{attribute 'OPC.UA.DA.StructuredType' := '1'}
{attribute 'OPC.UA.DA' := '1'}
TYPE stCombineAxisStatus :
STRUCT
    bEnabled : BOOL;
    bOperational : BOOL;
    bMoving : BOOL;
    bHomed : BOOL;
    bInSavePosition : BOOL;
    fActualPosition : LREAL;
    fActualVelocity : LREAL;
    fTargetPosition : LREAL;
    fZeroPoint : LREAL;
    fSafePosition : LREAL;
    nCommandID : UINT;
    eCommandStatus : eProgress;
END_STRUCT
END_TYPE

(* stored: Version 1.1.0.1, ProductVersion 3.1.4026.18
   DUT stCombineAxisStatus: Id {01a86c1f-d923-468f-aa17-d769d2d0e6ad} *)
